INTERFACE I_LimSwStatus

{warning 'Add property implementation'}
PROPERTY LimBackward : BOOL
GET
END_GET
END_PROPERTY

{warning 'Add property implementation'}
PROPERTY LimForward : BOOL
GET
END_GET
END_PROPERTY

{warning 'Add property implementation'}
PROPERTY LimHome : BOOL
GET
END_GET
END_PROPERTY

PROPERTY MoveBackwardEnabled : BOOL
GET
END_GET
END_PROPERTY

PROPERTY MoveForwardEnabled : BOOL
GET
END_GET
END_PROPERTY

END_INTERFACE

(* stored: Version 1.1.0.1
   Itf I_LimSwStatus: Id {256e382d-89de-4efb-b391-22faa6fe67b6}
   Property LimBackward: Id {68b52e9f-1d3c-4df6-85ee-1ebe2f49d852}
   Get Get: Id {4c7c79fc-0544-43b9-8d7a-5c3a42781093}
   Property LimForward: Id {f99a068d-d094-4bba-9373-2cc78b4facdc}
   Get Get: Id {eb8ad37e-7bb6-42e3-8c99-52bef6ee8db0}
   Property LimHome: Id {f4f52156-2af5-4624-9556-441d2ccf866e}
   Get Get: Id {b851cfcd-dff8-43f8-8b4b-a29d1e05e648}
   Property MoveBackwardEnabled: Id {b4e7f086-2ef8-4485-be7e-4532b5db4264}
   Get Get: Id {9b0ef177-2451-44cd-bad6-e27eaa34b91b}
   Property MoveForwardEnabled: Id {c448b972-f646-4f09-a55d-f335dff878cb}
   Get Get: Id {63539f14-b019-40ce-9a44-701a06eafced} *)
